(* IEC 61131-3 sources: AXOpen/src/integrations/app/src/Examples/AXOpen.AxoContext, 1 file *)

(* ---- AxoContextExample.st ---- *)
USING AXOpen.Core;

//<Implementation>
    PROGRAM ProgramExample
        VAR
            MyContext : AxoContextExample;
        END_VAR

        MyContext.Run();

    END_PROGRAM
//</Implementation>

//<Declaration>
    {S7.extern=ReadWrite}
    CLASS PUBLIC AxoContextExample EXTENDS  AXOpen.Core.AxoContext
        METHOD PROTECTED OVERRIDE Main
            // Here goes all your logic for given AxoContext.
            ;
        END_METHOD
    END_CLASS
//</Declaration>
